// TIA Portal V17 export
// export: Created 2024-09-02T12:50:30.9910905Z, ExportSetting WithDefaults, DisplayName Totally Integrated Automation Portal, DisplayVersion V17, DisplayName TIA Portal Openness, DisplayVersion V17, DisplayName TIA Portal Version Control Interface, DisplayVersion V17, DisplayName STEP 7 Professional, DisplayVersion V17, DisplayName STEP 7 Safety, DisplayVersion V17, DisplayName WinCC Professional, DisplayVersion V17
TYPE "Desoutter_Input"
// stored: IsFailsafeCompliant false
   STRUCT
      StartCycle : Bool;   // The tool runs as long as the signal is on “1”. When the signal drops, the cycle stops.
      Direction : Bool;   // Activates the untightening direction mode of the spindle at the “Start cycle”.
      Reset : Bool;   // Reset station tightening reports, all cycles’ counters, saved barcode
      Error_Acknowlage : Bool;   // When the error acknowledgement option is activated in the station parameters, the start of the spindle is not authorized after a reject report. The “error acknowledgement” input must be validated (pulse) to let the spindle start again By activating the error acknowledge input, the reject report output is reseted.
      Spindel_Validation : Bool;   // Allows, or not, the start cycle of the spindle(s). The spindle validation input is only taken into consideration by the CVIxII if the spindle validation source is set in the station parameters.
      Spindel_Ver_Rev : Bool;   // Untightening validation is only controlled when “Spindle validation on reverse” option is activated in the station parameters.
      Synchro_IN : Bool;   // Used in conjunction with Synchro OUT output to synchronise the tightening cycle phases of several controllers (synchro waiting phase).
      External_Stop : Bool;   // When the external stop option is set in a cycle rundown speed, final speed or run reverse phase, the controller will stops the current phase and shifts to the next one as soon as the signal shifts to “1”.
      CycleMode : Byte;   // Binary coded 1-2-4-8 cycle selection.The Cycle number selection 00 to 15 is only taken into consideration by the CVIx II if the “Source of cycle number” is set to “I/O” in the station parameters.
      PART_ID : Array[1..32] of Char;
   END_STRUCT;
END_TYPE
